FUNCTION AddToStringArray : BOOL
VAR_IN_OUT
	arr : ARRAY[*] OF STRING; //must start from 0 index
END_VAR
VAR_INPUT
	newString : STRING;
END_VAR
VAR_OUTPUT
	numElements : DINT;
	nextIndex : DINT;
END_VAR
VAR
	i : DINT;
END_VAR

FOR i:=LOWER_BOUND(arr, 1) TO UPPER_BOUND(arr, 1) BY 1 DO	
	IF arr[i] = '' THEN
		arr[i] := newString;
		nextIndex := i + 1;
		AddToStringArray := TRUE;
		EXIT;
	END_IF
	
END_FOR

numElements := UPPER_BOUND(arr, 1) - LOWER_BOUND(arr, 1) + 1;

CleanStringsArray(arr := arr);

END_FUNCTION

(* stored: Version 1.1.0.1, ProductVersion 3.1.4024.11
   POU AddToStringArray: Id {62533109-713d-4adc-8713-a6fe80ca70e7}, SpecialFunc None *)
